TEXTLIST FormatoTabla
  0 = 'Sin seleccionar'
  1 = '170x170'
  2 = '200x650'
  3 = '300x150'
  4 = '300x300'
  5 = '30x30'
  6 = 'Ninguno de la lista'
   = ''
END_TEXTLIST

(* stored: Version 1.1.0.1, ProductVersion 3.1.4024.12
   TextList FormatoTabla: Id {6c498501-58b7-4108-9246-c925940edd3a} *)
